// SIMATIC S7-200 project (STEP 7-Micro/WIN), CPU 221 REL 01.10

ORGANIZATION_BLOCK 主程序:OB1
TITLE=程序注释
BEGIN
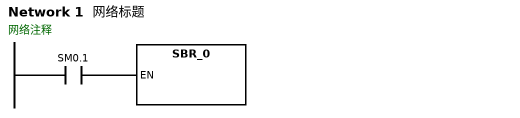
Network 1 // 网络标题
// 网络注释
// (network saved uncompiled; LAD cells follow)
// row 0: c0 -| |- SM0.1  c1 [SBR_0 EN:=power@row0]
END_ORGANIZATION_BLOCK

SUBROUTINE_BLOCK SBR_0:SBR0
TITLE=子程序注释
BEGIN
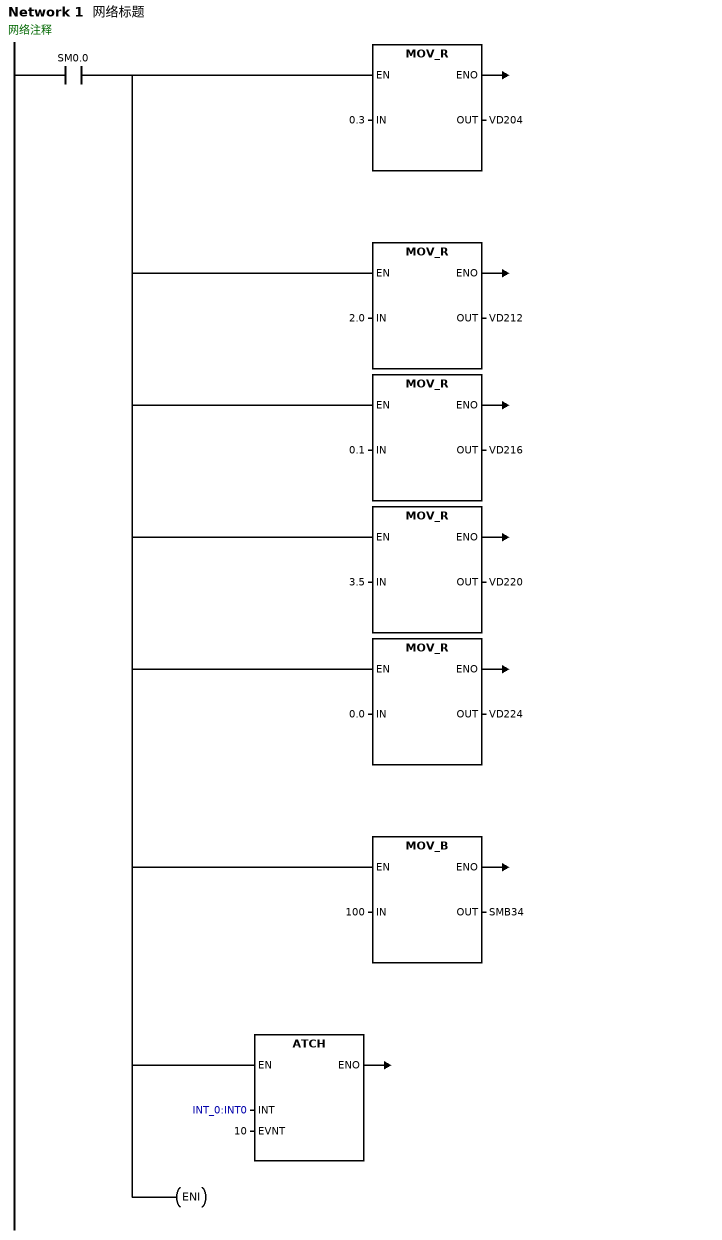
Network 1 // 网络标题
// 网络注释
// (network saved uncompiled; LAD cells follow)
// row 0: c0 -| |- SM0.0 v  c1 --  c2 --  c3 [MOV_R EN:=power@row0, IN:=0.3, ENO=>power, OUT=>VD204]  c4 ->
// row 1: c0 ^v  c3 [box]
// row 2: c0 ^v
// row 3: c0 ^v  c1 --  c2 --  c3 [MOV_R EN:=power@row3, IN:=2.0, ENO=>power, OUT=>VD212]  c4 ->
// row 4: c0 ^v  c3 [box]
// row 5: c0 ^v  c1 --  c2 --  c3 [MOV_R EN:=power@row5, IN:=0.1, ENO=>power, OUT=>VD216]  c4 ->
// row 6: c0 ^v  c3 [box]
// row 7: c0 ^v  c1 --  c2 --  c3 [MOV_R EN:=power@row7, IN:=3.5, ENO=>power, OUT=>VD220]  c4 ->
// row 8: c0 ^v  c3 [box]
// row 9: c0 ^v  c1 --  c2 --  c3 [MOV_R EN:=power@row9, IN:=0.0, ENO=>power, OUT=>VD224]  c4 ->
// row 10: c0 ^v  c3 [box]
// row 11: c0 ^v
// row 12: c0 ^v  c1 --  c2 --  c3 [MOV_B EN:=power@row12, IN:=100, ENO=>power, OUT=>SMB34]  c4 ->
// row 13: c0 ^v  c3 [box]
// row 14: c0 ^v
// row 15: c0 ^v  c1 --  c2 [ATCH EN:=power@row15, INT:=INT_0:INT0, EVNT:=10, ENO=>power]  c3 ->
// row 16: c0 ^v  c2 [box]
// row 17: c0 ^  c1 -(ENI)
END_SUBROUTINE_BLOCK

INTERRUPT_BLOCK INT_0:INT0
TITLE=中断程序注释
BEGIN
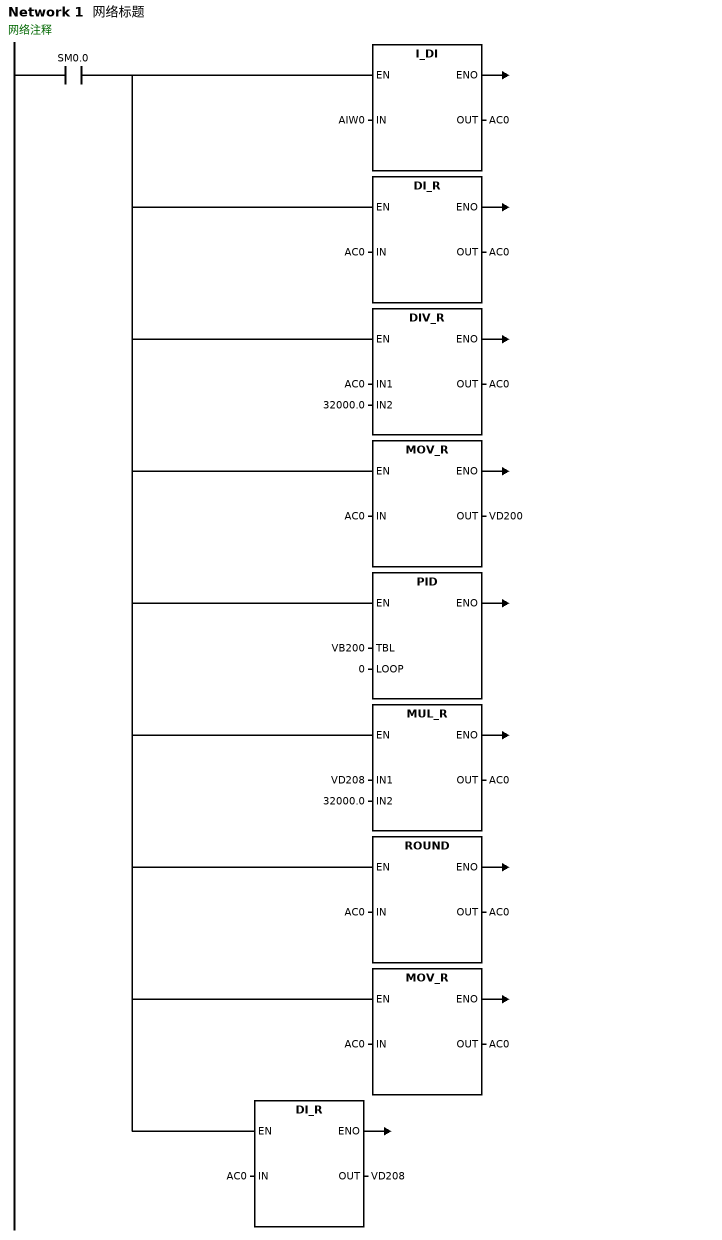
Network 1 // 网络标题
// 网络注释
// (network saved uncompiled; LAD cells follow)
// row 0: c0 -| |- SM0.0 v  c1 --  c2 --  c3 [I_DI EN:=power@row0, IN:=AIW0, ENO=>power, OUT=>AC0]  c4 ->
// row 1: c0 ^v  c3 [box]
// row 2: c0 ^v  c1 --  c2 --  c3 [DI_R EN:=power@row2, IN:=AC0, ENO=>power, OUT=>AC0]  c4 ->
// row 3: c0 ^v  c3 [box]
// row 4: c0 ^v  c1 --  c2 --  c3 [DIV_R EN:=power@row4, IN1:=AC0, IN2:=32000.0, ENO=>power, OUT=>AC0]  c4 ->
// row 5: c0 ^v  c3 [box]
// row 6: c0 ^v  c1 --  c2 --  c3 [MOV_R EN:=power@row6, IN:=AC0, ENO=>power, OUT=>VD200]  c4 ->
// row 7: c0 ^v  c3 [box]
// row 8: c0 ^v  c1 --  c2 --  c3 [PID EN:=power@row8, TBL:=VB200, LOOP:=0, ENO=>power]  c4 ->
// row 9: c0 ^v  c3 [box]
// row 10: c0 ^v  c1 --  c2 --  c3 [MUL_R EN:=power@row10, IN1:=VD208, IN2:=32000.0, ENO=>power, OUT=>AC0]  c4 ->
// row 11: c0 ^v  c3 [box]
// row 12: c0 ^v  c1 --  c2 --  c3 [ROUND EN:=power@row12, IN:=AC0, ENO=>power, OUT=>AC0]  c4 ->
// row 13: c0 ^v  c3 [box]
// row 14: c0 ^v  c1 --  c2 --  c3 [MOV_R EN:=power@row14, IN:=AC0, ENO=>power, OUT=>AC0]  c4 ->
// row 15: c0 ^v  c3 [box]
// row 16: c0 ^  c1 --  c2 [DI_R EN:=power@row16, IN:=AC0, ENO=>power, OUT=>VD208]  c3 ->
// row 17: c2 [box]
END_INTERRUPT_BLOCK
